INTERFACE ITF_Cyclic

METHOD CyclicUpdate : BOOL
VAR_INPUT
END_VAR
END_METHOD

END_INTERFACE

(* stored: Version 1.1.0.1
   Itf ITF_Cyclic: Id {ed9f9542-9ab5-4a80-9c5e-5b531721665e}
   Method CyclicUpdate: Id {f69038f0-99c9-4f02-8d55-1fa5beb2505d} *)
